FUNCTION_BLOCK RunUnitControllerV1 EXTENDS RunUnitGeneric
VAR_INPUT
END_VAR
VAR_OUTPUT
	currentMode : eOperationModes := eOperationModes.MANUAL; //default in semi-auto
	isInitializing : BOOL;
	isError : BOOL;
	
END_VAR
VAR		
	nCounter : INT;
	bAllInitialized : BOOL := FALSE;
	
	//user control
	requestInitialize : BOOL;
	//error
	requestErrorClear : eErrorClearWays := eErrorClearWays.NO_ACTION;
	errorDevice : POINTER TO CommonBase := 0; //null reference
	errorType : eCategrories;
	errorIndex : INT;
	errorCode : UDINT;
	errorDelayDetect : TON;	
	//HMI Control interface
	interfaceControl : POINTER TO InterfaceControlV1;
	interfaceManual : POINTER TO InterfaceManualV1;
	
	pbRed : POINTER TO RunSignal;
	pbGreen : POINTER TO RunSignal;
	pbYellow : POINTER TO RunSignal;
END_VAR
VAR PERSISTENT
	axisUpperBound : INT;
	cylinderUpperBound : INT;
	signalUpperBound : INT;
	unitUpperBound : INT;
	slotUpperBound : int;
END_VAR

//scan running all devices
FOR nCounter :=1 TO axisUpperBound BY 1 DO
	gvl.axisControls[nCounter]();
	//error detection
	IF errorDevice=0 AND errorDelayDetect.Q AND gvl.axisControls[nCounter].ErrorDetect() <> 0 THEN
		//error scaned
		interfaceControl^.errorIndex := TO_DWORD(nCounter-1);
		errorDevice := ADR(gvl.axisControls[nCounter]);
	END_IF
END_FOR
FOR nCounter :=1 TO cylinderUpperBound BY 1 DO
	gvl.cylinderControls[nCounter]();
	//error detection
	IF errorDevice=0 AND errorDelayDetect.Q AND gvl.cylinderControls[nCounter].ErrorDetect() <> 0 THEN
		//error scaned
		interfaceControl^.errorIndex := TO_DWORD(nCounter-1);
		errorDevice := ADR(gvl.cylinderControls[nCounter]);
	END_IF
END_FOR
FOR nCounter :=1 TO signalUpperBound BY 1 DO
	gvl.signalControls[nCounter]();
END_FOR
FOR nCounter :=1 TO unitUpperBound BY 1 DO
	//error detection
	IF errorDevice=0 AND errorDelayDetect.Q AND gvl.units[nCounter] <> 0 AND_THEN gvl.units[nCounter]^.ErrorDetect() <> 0THEN
		//station
		interfaceControl^.errorIndex := TO_DWORD(nCounter-1);
		errorDevice := gvl.units[nCounter];
	END_IF
END_FOR
//routines
errorDelayDetect(IN:= (errorDevice = 0), PT:= T#100MS, Q=> , ET=> );	//after reset , wait 100ms to detect
IF errorDevice <>0 THEN
	//errorIndex := nCounter-1;
	interfaceControl^.errorType := errorDevice^.TypeCode();
	interfaceControl^.errorCode := errorDevice^.ErrorDetect();
		
	ErrorHandler();// handling user-input reset/ignore
ELSE
	//reset
	interfaceControl^.errorType := 0;
	interfaceControl^.errorIndex := 0;
	interfaceControl^.errorCode := 0;
END_IF
isError := errorDevice <>0;
//reflect to interface
interfaceManual^(
	currentMode:= THIS^.currentMode); //scan-in,scan-out,manual...
//handling input request
interfaceControl^(
	currentMode:= THIS^.currentMode,
	pbGreen := pbGreen^.debouncedOn,
	pbRed := pbRed^.debouncedOn,
	pbYellow := pbYellow^.debouncedOn,
	errorClear=> THIS^.requestErrorClear);
IF interfaceControl^.requestInit THEN
	requestInitialize := TRUE; // memorize
END_IF
//mode switcher pre-check
bPause := NOT (currentMode = eOperationModes.AUTO);
IF interfaceControl^.requestMode <> currentMode THEN
	CASE interfaceControl^.requestMode OF 
		eOperationModes.MANUAL,eOperationModes.SEMI_AUTO:
			//direct changes
			currentMode := interfaceControl^.requestMode;
		eOperationModes.AUTO:
			//check : no error , manual channel work done
			IF errorDevice=0 THEN
				currentMode := eOperationModes.AUTO;
			ELSE
				//refuce to change , maintain
			END_IF 
	END_CASE
END_IF
//
CASE currentMode OF	
		eOperationModes.AUTO,eOperationModes.SEMI_AUTO:
		//running sequences
		FOR nCounter :=1 TO unitUpperBound BY 1 DO
			IF gvl.units[nCounter] <> 0 THEN
				gvl.units[nCounter]^();
			END_IF
		END_FOR
		
		IF  requestInitialize THEN
			//initialize all stations
			bAllInitialized := TRUE;
			interfaceControl^.state := TO_WORD(eSpecialStates.MAIN_INITIALIZING); //status reflection
			
			FOR nCounter:=1 TO unitUpperBound BY 1 DO
				IF gvl.units[nCounter] <> 0 THEN
					// if every station comes initialized
					bAllInitialized := bAllInitialized AND gvl.units[nCounter]^.Initialize();
				END_IF
			END_FOR
			IF bAllInitialized THEN
				FOR nCounter:=1 TO unitUpperBound BY 1 DO
					IF gvl.units[nCounter] <> 0 THEN
						gvl.units[nCounter]^.NextState := 0; //start working
					END_IF
				END_FOR	
				requestInitialize := FALSE; //clear after done
				//---------------------------------
				//	Clear all material valid status
				//---------------------------------
				FOR nCounter:=1 TO slotUpperBound BY 1 DO
					gvl.materialSlots[nCounter].Valid := FALSE;
				END_FOR
				
				interfaceControl^.state := TO_WORD(eSpecialStates.MAIN_INITIALIZED); //status reflection
			END_IF
		END_IF		
END_CASE

//status reflect
isInitializing := requestInitialize AND NOT bAllInitialized;
//

METHOD ErrorHandler : BOOL
VAR_INPUT
END_VAR
VAR
END_VAR
//once error scanned
IF currentMode = eOperationModes.AUTO THEN
	//once error deteted and in AUTO mode , forcely switch to SEMI_AUTO
	currentMode := eOperationModes.SEMI_AUTO;
END_IF
//reset error handling
IF requestErrorClear <> eErrorClearWays.NO_ACTION THEN
	errorDevice^.ErrorClear(requestErrorClear); //call error clear function
	requestErrorClear := eErrorClearWays.NO_ACTION;
	errorDevice := 0 ;// cut link
END_IF
END_METHOD

METHOD FB_init : BOOL
VAR_INPUT
	bInitRetains : BOOL; // if TRUE, the retain variables are initialized (warm start / cold start)
	bInCopyCode : BOOL;  // if TRUE, the instance afterwards gets moved into the copy code (online change)
	
	argParent : POINTER TO RunUnitGeneric;
	argSlotBase : POINTER TO RunMaterial;
	argSlotLast : POINTER TO RunMaterial;
	
	argPbRed : POINTER TO RunSignal;
	argPbGreen : POINTER TO RunSignal;
	argPbYellow : POINTER TO RunSignal;
	
	argInterfaceControl : POINTER TO InterfaceControlV1;
	argInterfaceManual : POINTER TO InterfaceManualV1;
END_VAR
//initialize 
Parent := argParent;
SlotBase := argSlotBase;
SlotLast := argSlotLast;
//
IF bInitRetains THEN
	NextState := eSpecialStates.INITIAL_BEGIN;
END_IF
//input
pbRed := argPbRed;
pbGreen := argPbGreen;
pbYellow := argPbYellow;

interfaceControl := argInterfaceControl;
interfaceManual := argInterfaceManual;

interfaceControl^.state := TO_WORD(eSpecialStates.MAIN_WAIT_INITIALIZING);
END_METHOD

METHOD Initialize : BOOL
VAR_INPUT
END_VAR
END_METHOD

END_FUNCTION_BLOCK

(* stored: Version 1.1.0.1, ProductVersion 3.1.4024.0
   POU RunUnitControllerV1: Id {dbefb355-befd-4ccc-b7d8-49a15cbd5d5f}, SpecialFunc None
   Method ErrorHandler: Id {a0eb5aec-6465-4175-9953-8d5b0f3a2dc2}
   Method FB_init: Id {1060438f-10b7-4590-a96e-41200ea3be54}
   Method Initialize: Id {cb68dc91-f1ca-48a3-a360-7027131d9307} *)
